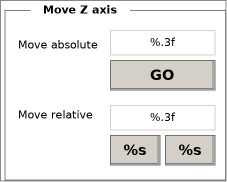
VISUALIZATION VISU_M2ZAxisControl  // 227x182
VAR_IN_OUT
	widget : M2AxisWidget;
END_VAR
    Label (40,0 140x20), "Move Z axis"
    Polyline (130,10) (225,10) (225,180) (5,180) (5,10) (30,10)
    Textfield (110,30 105x25), "%.3f", text variable: widget.absolute_setpoint
        OnMouseClick: write the text variable via VisuDialogs.Numpad, title 'Enter the absolute position setpoint in mm'
    Textfield (110,105 105x25), "%.3f", text variable: widget.relative_setpoint
        OnMouseClick: write the text variable via VisuDialogs.Numpad, title 'Enter the relative position offset in mm'
    Button (110,60 105x30), "GO", input disabled if: widget.absolute_go_disabled
        OnMouseClick: execute { widget.absolute_go := TRUE; }
    Button (110,135 50x30), "%s", text variable: widget.relative_goLeft_text, input disabled if: widget.relative_goLeft_disabled
        OnMouseClick: execute { widget.relative_goLeft := TRUE; }
    Button (165,135 50x30), "%s", text variable: widget.relative_goRight_text, input disabled if: widget.relative_goRight_disabled
        OnMouseClick: execute { widget.relative_goRight := TRUE; }
    Label (15,30 90x30), "Move absolute"
    Label (15,100 90x30), "Move relative"
END_VISUALIZATION

(* stored: Version 1.1.0.1, ProductVersion 3.1.4018.5
   Visu VISU_M2ZAxisControl: Id {69926236-cfd1-46ce-a1a2-da23d1acbc96} *)
